FUNCTION_BLOCK CROSSCOMM_SENDER_271612CFD7010AE0 (* Service Interface Function Block Type *)
  (* Standard: 61499-2 *)
  (* Version 0.0, 9/22/2017, bababen, nxtControl GmbH, template *)
  PACKAGE Main;
  (* Compiler Cpp nxtControl builtin 1.0 *)
  {SET_ATTRIBUTE(Runtime.FBType.ImplementingType, Runtime.System#DYNGEN_CROSSCOMM_SENDER)}
  {SET_ATTRIBUTE(Configuration.GenericFBType.InterfaceParams, Runtime.System#<InterfaceList> <EventInputs> <Event Name="INITO" /> <Event Name="CNF"> <With Var="ExtendPusher" /> </Event> </EventInputs> <InputVars> <VarDeclaration Name="ExtendPusher" Type="BOOL" /> </InputVars> </InterfaceList>)}
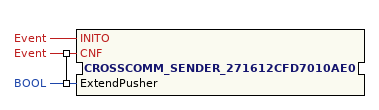
  EVENT_INPUT
    INITO;
    CNF WITH ExtendPusher;
  END_EVENT
  VAR_INPUT
    ExtendPusher : BOOL;
  END_VAR
  EC_STATES
    START;
  END_STATES
END_FUNCTION_BLOCK
